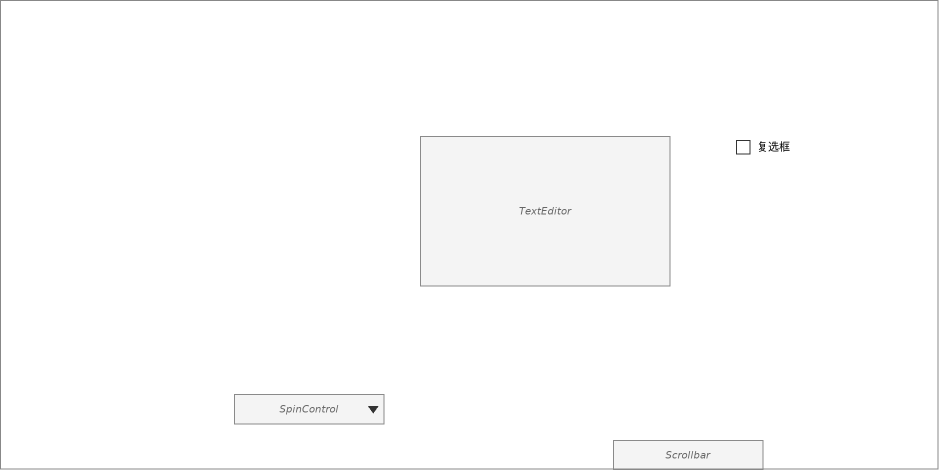
VISUALIZATION Visualization  // 939x470
    TextEditor (420,136 250x150)
        p4127561890: Courier New
    Scrollbar (613,440 150x30)
    InvisibleInput (789,270 150x30)
    SpinControl (234,394 150x30)
        OnMouseDown: write UserMode.UserGapPositionNew via Default
    Checkbox (734,132 150x30), "复选框"
END_VISUALIZATION

(* stored: Version 1.1.0.1, ProductVersion 3.1.4024.6
   Visu Visualization: Id {80a43d98-2052-4fe5-a39d-f1ab323d2ecb} *)
